# EPICS substitutions: db/ecmcFIODrive_DRV.substitutions
# All fields related to velocity scaling and alarms
file ecmcFIODrive_DRV.template
{
	pattern {LINR,    ESLO,   EOFF,   EGU,        PREC, LOW, LOLO, HIGH, HIHI, HYST, LLSV,       LSV,        HSV,        HHSV      }
		{"SLOPE", 1,      0,      "Raw",      0,    0,   0,    0,    0,    0,    "NO_ALARM", "NO_ALARM", "NO_ALARM", "NO_ALARM"}
}
